TEXTLIST TextList_01
   = ''
END_TEXTLIST

(* stored: Version 1.1.0.1
   TextList TextList_01: Id {2a7013b7-81d8-0450-19f0-a978cab3e43d} *)
